// Mitsubishi GX Works2 project: q5   PLC: Q02/Q02H

PROGRAM MAIN
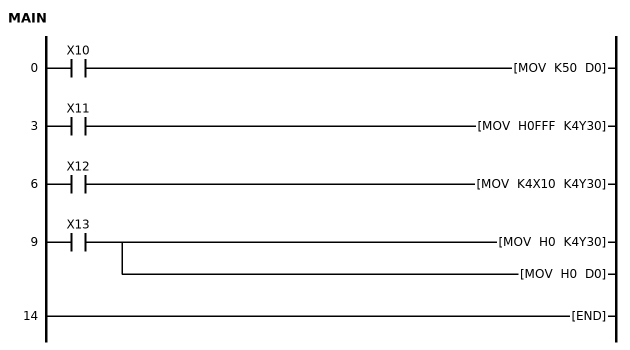
0     LD      X10
      MOV     K50 D0
3     LD      X11
      MOV     H0FFF K4Y30
6     LD      X12
      MOV     K4X10 K4Y30
9     LD      X13
      MOV     H0 K4Y30
      MOV     H0 D0
14    END
END_PROGRAM
